INTERFACE ITF_Control2_HMI_Connector_View EXTENDS ITF_BaseControlElement_HMI_Connector_View

END_INTERFACE

(* stored: Version 1.1.0.1
   Itf ITF_Control2_HMI_Connector_View: Id {f58443bb-275f-050c-0d32-569d8b0a37aa} *)
